FUNCTION F_ConfigExternalDestination : BOOL



;

END_FUNCTION

(* stored: Version 1.1.0.1, ProductVersion 3.1.4024.9
   POU F_ConfigExternalDestination: Id {f56759ed-2a31-4a2b-b4cc-47283f0eba82}, SpecialFunc None *)
